TYPE T_Ctrl_SIf_MOD_Cfg :
STRUCT
	/// Enable communication to line control
	bolComToLineControlEnabled: BOOL;
	/// Ignore Ready Input
	bolIgnoreReadyInput: BOOL;
	/// True = Enable the Stacklight Horn
	bolStackLightHornEnable: BOOL;
END_STRUCT
END_TYPE

(* stored: Version 1.1.0.1, ProductVersion 3.1.0.36
   DUT T_Ctrl_SIf_MOD_Cfg: Id {0a6ad749-9fa3-41c0-ba6b-a045ebbc52d5} *)
